(* CODESYS project WAGO.export

Project tree, tasks and I/O mapping:
  Switches/
    function block Direct [ST]: xLamp
    function block Latch [ST]: xLamp
  interface ITF01: xLamp
  program PLC_PRG [ST]
  visualisation Visualization
*)

// ITF01
INTERFACE ITF01

METHOD xLamp : BOOL
VAR_INPUT
	xSwitch	: BOOL;
END_VAR
END_METHOD

END_INTERFACE

// PLC_PRG
PROGRAM PLC_PRG
VAR
	D01	: Direct;
	L01	: Latch;

	xLight	: BOOL;
	xSwitch	: BOOL;
END_VAR

xLight := L01.xLamp(xSwitch := xSwitch);

END_PROGRAM

// Switches/Direct
FUNCTION_BLOCK Direct IMPLEMENTS ITF01
VAR_INPUT
END_VAR
VAR_OUTPUT
END_VAR
VAR
END_VAR

{warning 'add method implementation '}
METHOD xLamp : BOOL
VAR_INPUT
	xSwitch	: BOOL;
END_VAR
xLamp := xSwitch;
END_METHOD

END_FUNCTION_BLOCK

// Switches/Latch
FUNCTION_BLOCK Latch IMPLEMENTS ITF01
VAR_INPUT
END_VAR
VAR_OUTPUT
END_VAR
VAR
	_xBuffer : BOOL;
	_trigger : R_TRIG;
END_VAR

{warning 'add method implementation '}
METHOD xLamp : BOOL
VAR_INPUT
	xSwitch	: BOOL;
END_VAR
_trigger(CLK := xSwitch);

IF (_trigger.Q) THEN
	_xBuffer := NOT _xBuffer;
END_IF

xLamp := _xBuffer;
END_METHOD

END_FUNCTION_BLOCK

// /Visualization
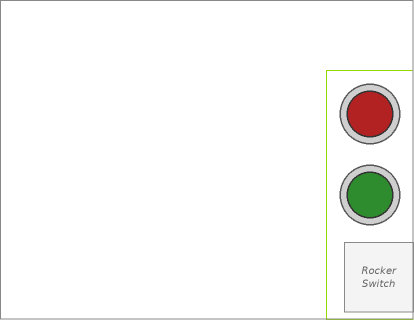
VISUALIZATION Visualization  // 414x320
    RoundedRectangle (326,70 87x250)
    Lamp1 (335,79 70x70), variable: NOT PLC_PRG.xLight, style: Lamp-Lamp1-Red
    RockerSwitch (344,242 70x70), variable: PLC_PRG.xSwitch, behaviour: TOGGLE, style: Switch-RockerSwitch-Gray
    Lamp1 (335,160 70x70), variable: PLC_PRG.xLight, style: Lamp-Lamp1-Green
END_VISUALIZATION
